{attribute 'qualified_only'}
{attribute 'strict'}
{attribute 'to_string'}
TYPE eSystemCommand :
(
	KEINE		:= 0,
	AUSCHALTEN 	:= 1,
	EINSCHALTEN := 2,
	STOPPEN		:= 3,
	RESETTEN	:= 4
);
END_TYPE

(* stored: Version 1.1.0.1
   DUT eSystemCommand: Id {b681ae9b-183a-458d-837e-9a7c35584e58} *)
